// TIA Portal V17 export
// export: Created 2024-08-07T21:44:17.7010291Z, ExportSetting WithDefaults, DisplayName Totally Integrated Automation Portal, DisplayVersion V17 Update 7, DisplayName TIA Portal Openness, DisplayVersion V17 Update 7, DisplayName TIA Portal Version Control Interface, DisplayVersion V17, DisplayName SINAMICS Startdrive Advanced, DisplayVersion V17 SP2, DisplayName SINAMICS Startdrive G110M, G120, G120C, G120D, G120P, G115D, DisplayVersion V17 SP2, DisplayName SINAMICS Startdrive G130, G150, S120, S150, SINAMICS MV, S210, DisplayVersion V17 SP2, DisplayName STEP 7 Professional, DisplayVersion V17 Update 7, DisplayName STEP 7 Safety, DisplayVersion V17 Update 6, DisplayName WinCC Advanced / Unified PC, DisplayVersion V17 Update 7
TYPE "typeOpcUaJIG"
// stored: IsFailsafeCompliant false
   STRUCT
      Clamping_Step_Round1 : Int;
      Clamping_Step_Round2 : Int;
      Initialize : Bool;
      InLoading : Bool;
      Jig_Clamped : Bool;
      Jig_Error : Int;
      Jig_ID : USInt;
      Jig_Loading_Position : Bool;
      Jig_Unclamped : Bool;
      Part_In : Bool;
      Part_NOK : Bool;
      Part_OK : Bool;
      Positioner_Operator_Position : Bool;
      Product_ID : USInt;
      Product_Out : Bool;
      Request_Door_Closing : Bool;
      Request_Door_Opening : Bool;
      Start_Clamping : Bool;
      Start_Unclamping : Bool;
      TimestampJIG : LDT;
      Unclamping_Step_Round1 : Int;
      Unclamping_Step_Round2 : Int;
      Wait_Start : Bool;
      WeldStageNumber : USInt;
   END_STRUCT;
END_TYPE
